FUNCTION_BLOCK PIDController
  (* Standard: 61499-2 *)
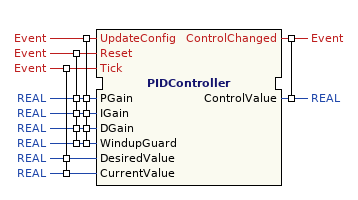
  EVENT_INPUT
    UpdateConfig WITH PGain, IGain, DGain, WindupGuard;
    Reset WITH PGain, IGain, DGain, WindupGuard;
    Tick WITH DesiredValue, CurrentValue;
  END_EVENT
  EVENT_OUTPUT
    ControlChanged WITH ControlValue;
  END_EVENT
  VAR_INPUT
    PGain : REAL;
    IGain : REAL;
    DGain : REAL;
    WindupGuard : REAL;
    DesiredValue : REAL;
    CurrentValue : REAL;
  END_VAR
  VAR_OUTPUT
    ControlValue : REAL;
  END_VAR
  VAR
    pTerm : REAL;
    iTerm : REAL;
    dTerm : REAL;
    previousError : REAL;
    currentError : REAL;
    integrationError : REAL;
    differentialError : REAL;
  END_VAR
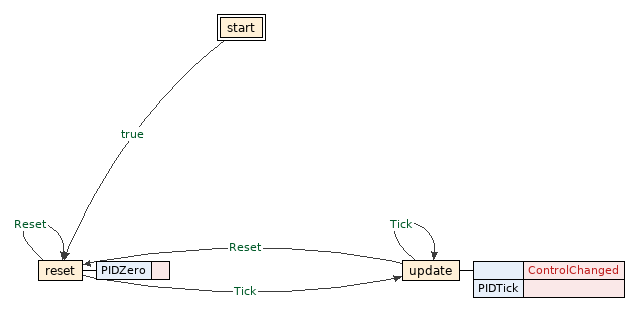
  EC_STATES
    start;
    update : -> ControlChanged, PIDTick;
    reset : PIDZero;
  END_STATES
  EC_TRANSITIONS
    start TO reset := true;
    update TO reset := Reset;
    update TO update := Tick;
    reset TO reset := Reset;
    reset TO update := Tick;
  END_TRANSITIONS
  ALGORITHM PIDTick IN ST:
        //calculate proportional error
        currentError := DesiredValue - ActualValue;

        //calculate integrationError (with WindupGuard clamp)
        integrationError += currentError;
        if integrationError < -WindupGuard then
            integrationError := -WindupGuard;
        elsif integrationError > -WindupGuard then
            integrationError := WindupGuard;
        end_if;

        //calculate differentation error
        differentialError := currentError - previousError;

        // scaling
        pTerm := PGain * currentError;
        iTerm := IGain * integrationError;
        dTerm := DGain * differentialError;

        // output the summation of terms
        Control := pTerm + iTerm + dTerm;

        // save current error as previous error for next iteration
        previousError = currentError;
  END_ALGORITHM
  ALGORITHM PIDZero IN ST:
        //reset the only persistent internal variables to zero the PID
        previousError := 0;
        integrationError := 0;
  END_ALGORITHM
END_FUNCTION_BLOCK
